Fanuc KAREL source: kt00220.KL

-- PROVISIONAL review KL for V770-1; original PC SHA256 dbfd7bef3ff3975f2e66357d4f3e2682da45e413f44dad14f6a70336377b87fc
-- Incomplete behavior may be omitted. Consult companion uncertainty JSON. Do not deploy.
PROGRAM KT00220
%NOLOCKGROUP
VAR
  I2 : INTEGER
  OUT : INTEGER
-- UNRESOLVED_DECL H1 type=002017
BEGIN
  -- UNRESOLVED_PC offsets 5-19; opcodes 2E,22,9D,33,B4
  -- UNRESOLVED_PC offsets 24-35; opcodes 2E,23
  -- UNRESOLVED_PC offsets 40-62; opcodes 22,9D,33,B3,21,46,23
  -- UNRESOLVED_PC offsets 67-71; opcodes 7F
END KT00220
